{attribute 'OPC.UA.DA' := '0'}
TYPE PolarisationConfig :
STRUCT
	PolarAngle_S : LREAL;
	PolarAngle_P : LREAL;
END_STRUCT
END_TYPE

(* stored: Version 1.1.0.1, ProductVersion 3.1.4024.3
   DUT PolarisationConfig: Id {a2b49a86-0d1a-4bf2-9947-976db2a0edb5} *)
